FUNCTION_BLOCK INI_AIS (* Load and Store STRING Data from settings.ini by Section and Key (AIS Adapter Interface) *)
  (* Standard: 61499-2; Description: Copyright (c) 2026 Meisterschulen am Ostbahnhof This program and the accompanying materials are made available under the terms of the Eclipse Public License 2.0 which is available at https://www.eclipse.org/legal/epl-2.0/ SPDX-License-Identifier: EPL-2.0 *)
  (* Version 1.0, 2026-04-13, Franz Höpfinger, Meisterschulen am Ostbahnhof, initial API and implementation and/or initial documentation *)
  PACKAGE eclipse4diac::storage;
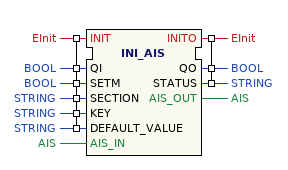
  EVENT_INPUT
    INIT : EInit WITH QI, SETM, SECTION, KEY, DEFAULT_VALUE; (* Service Initialization *)
  END_EVENT
  EVENT_OUTPUT
    INITO : EInit WITH QO, STATUS; (* Initialization Confirm *)
  END_EVENT
  VAR_INPUT
    QI : BOOL; (* Event Input Qualifier *)
    SETM : BOOL; (* Enable Mirroring on SET *)
    SECTION : STRING; (* Section name. *)
    KEY : STRING; (* Key name. *)
    DEFAULT_VALUE : STRING; (* The value to read if there is nothing in the settings.ini *)
  END_VAR
  VAR_OUTPUT
    QO : BOOL; (* Event Output Qualifier *)
    STATUS : STRING; (* Service Status *)
  END_VAR
  SOCKETS
    AIS_IN : adapter::types::unidirectional::AIS; (* Value to store (SET) *)
  END_SOCKETS
  PLUGS
    AIS_OUT : adapter::types::unidirectional::AIS; (* Stored value output (GETO) *)
  END_PLUGS
  FBS
    INI : eclipse4diac::storage::INI;
    SET_PERMIT : iec61499::events::E_PERMIT;
  END_FBS
  EVENT_CONNECTIONS
    INIT TO INI.INIT;
    INI.INITO TO INITO;
    INI.INITO TO INI.GET;
    AIS_IN.E1 TO INI.SET;
    INI.GETO TO AIS_OUT.E1;
    SET_PERMIT.EO TO AIS_OUT.E1;
    INI.SETO TO SET_PERMIT.EI;
  END_CONNECTIONS
  DATA_CONNECTIONS
    QI TO INI.QI;
    SETM TO SET_PERMIT.PERMIT;
    SECTION TO INI.SECTION;
    KEY TO INI.KEY;
    DEFAULT_VALUE TO INI.DEFAULT_VALUE;
    AIS_IN.D1 TO INI.VALUE;
    INI.VALUEO TO AIS_OUT.D1;
    INI.QO TO QO;
    INI.STATUS TO STATUS;
  END_CONNECTIONS
END_FUNCTION_BLOCK
